TYPE ACRMemoryRealEvent EXTENDS ACRMemoryEvent :
STRUCT
	_Value : REAL;
END_STRUCT
END_TYPE

(* stored: Version 1.1.0.1, ProductVersion 3.1.4020.12
   DUT ACRMemoryRealEvent: Id {31f24b9a-b2c4-412b-b276-0697a3ac87e5} *)
